(* PLC project motors, Dassault Systèmes ControlBuild 2024x Refresh1 *)
(* stored: creationDateTime 2024-04-09T15:09:06-01:00 *)

FUNCTION_BLOCK flask_motion_app.motors
  VAR_INPUT
    Auto : BOOL := false;
    Manu : BOOL := false;
    run : BOOL := false;
  END_VAR
  VAR_INPUT
    presConvUp : BOOL := false;
    presConvDw : BOOL := false;
    masterPosition : REAL := 0.0;
    mesuredWeight : INT := 0;
  END_VAR
  VAR_INPUT
    phaseCode : INT := 0;
  END_VAR
  VAR_OUTPUT
    forwardUp : BOOL := false;
    backwardUp : BOOL := false;
  END_VAR
  VAR_OUTPUT
    forwardDw : BOOL := false;
    backwardDw : BOOL := false;
  END_VAR
  VAR_OUTPUT
    ejectBadProd : BOOL := false;
    weihtOk : BOOL := false;
  END_VAR
  VAR
    upperLimitOk : BOOL := false;
    lowerLimitOk : BOOL := false;
  END_VAR
  VAR CONSTANT
    prtSensorConvDw : TIME := T#0h0m0s500ms;
    prtSensorConvUp : TIME := T#0h0m0s800ms;
    upperLimitWeight : INT := 125;
    lowerLimitWeight : INT := 115;
  END_VAR

(* LD diagram, written out as Structured Text *)
1:
le_int1(IN0 := mesuredWeight, IN1 := upperLimitWeight);
upperLimitOk := le_int1.OUT;
gt_int1(IN0 := mesuredWeight, IN1 := lowerLimitWeight);
lowerLimitOk := gt_int1.OUT;
weihtOk := upperLimitOk AND lowerLimitOk;
ton1(IN := Auto AND run AND NOT presConvDw, PT := prtSensorConvUp);
backwardDw := ton1.Q;
tof1(IN := ?, PT := prtSensorConvDw);
forwardUp := tof1.Q;
ejectBadProd := Auto AND run AND presConvDw AND NOT weihtOk AND NOT backwardDw;
(* drawn but not wired to any output: Auto, run, presConvUp *)
END_FUNCTION_BLOCK
